Fanuc KAREL source: MP0082.KL

PROGRAM MP0082
%STACKSIZE=65535
%PRIORITY=65535
%NOLOCKGROUP
ROUTINE FINT(P1 : INTEGER) : INTEGER FROM MP0082
ROUTINE FREAL(P1 : REAL) : REAL FROM MP0082
ROUTINE RTEST(P1 : INTEGER; P2 : REAL) FROM MP0082
ROUTINE FINT
BEGIN
-- UNRESOLVED_PC line 5 opcodes [2D 9D 52 7F] marker_code=1
-- UNRESOLVED_PC line 6 opcodes [7F] marker_code=18
END FINT
ROUTINE FREAL
BEGIN
-- UNRESOLVED_PC line 9 opcodes [2D 2E 69 7F] marker_code=28
-- UNRESOLVED_PC line 10 opcodes [7F] marker_code=49
END FREAL
ROUTINE RTEST
VAR
L1 : ARRAY[3] OF REAL
U2C_5 : INTEGER -- ASSUMED 2C source type; see uncertainty report
U2C_6 : INTEGER -- ASSUMED 2C source type; see uncertainty report
U2C_7 : INTEGER -- ASSUMED 2C source type; see uncertainty report
U2C_8 : INTEGER -- ASSUMED 2C source type; see uncertainty report
U2C_9 : INTEGER -- ASSUMED 2C source type; see uncertainty report
U2C_10 : INTEGER -- ASSUMED 2C source type; see uncertainty report
U2C_11 : REAL -- ASSUMED 2C source type; see uncertainty report
S1 : REAL
BEGIN
U2C_5=7
U2C_6=3
U2C_7=2
U2C_8=1075838976
U2C_9=1083179008
U2C_10=1069547520
L1[1]=2.5
S1=(L1[1] / U2C_9)
END RTEST
BEGIN
RTEST(7,2.5)
END MP0082
